FUNCTION_BLOCK SequenceTask EXTENDS TcoCore.TcoTask
VAR_INPUT
    Sequence : TcoCore.ITcoSequencer;
END_VAR

(*~
    <docu>
        <summary>
            Restores this instance to the Ready state. Can be called explicitly or from within one of the restore mechanisms.
            <para>
                See also <see cref="PlcDocu.TcoCore.TcoTask.AutoRestorable()"/>
            </para>
        </summary>
    </docu>
~*)
METHOD Restore : ITcoRestorable
SUPER^.Restore();
THIS^.Sequence.Restore();
END_METHOD

END_FUNCTION_BLOCK

(* stored: Version 1.1.0.1, ProductVersion 3.1.4024.12
   POU SequenceTask: Id {2fbae23c-7e65-0276-292f-a17539f73f10}, SpecialFunc None
   Method Restore: Id {abe851eb-8518-091f-33d8-c6ee8b69201a} *)
